{attribute 'GeneratedUsingTerminal: EL6224-0090-0016'}
{attribute addProperty BoxType "EL6224-0090-0016"}
{attribute addProperty Id "DeviceState_Inputs_DeviceDeviceState_Inputs_Device_A12105982"}
{attribute addProperty CRC "1394749468"}
{attribute addProperty Size "2"}
TYPE Module_1_DeviceState_Inputs_Device_5322301C :
STRUCT
	{attribute addProperty Name "DeviceState_Inputs_Device"}
	DeviceState_Inputs_Device  : DeviceState_Inputs_Device_A1210598;
END_STRUCT
END_TYPE

(* stored: Version 1.2.0.0, ProductVersion 3.1.4024.9
   DUT Module_1_DeviceState_Inputs_Device_5322301C: Id {3a120866-9214-487a-8a11-80494a81a772} *)
